// TwinCAT 3 PLC project PackML_Base
// ProgramVersion: 3.1.4023.0
// libraries:
//   PackML State Machine, * (ChrisK)
//   State Pattern PackML, * (ChrisK)
//   Tc2_Standard, * (Beckhoff Automation GmbH)
//   Tc2_System, * (Beckhoff Automation GmbH)
//   Tc3_Module, * (Beckhoff Automation GmbH)
//   Tc3_PackML_V2, * (Beckhoff Automation GmbH)
// project tree:
//   PackML_Method_Sample/ PML_Method_Sample.TcPOU
//   PackML_State_Sample/ Execute_State_Sample.TcPOU, PML_Sample_Class.TcPOU (not stored), Resetting_State_Sample.TcPOU, Starting_State_Sample.TcPOU
//   / PlcTask.TcTTO
//   POUs/ MAIN.TcPOU
// real-time tasks:
//   TASK PlcTask: cycle T#10ms, priority 20, ADS port 350

CONFIGURATION PackML_Base
    RESOURCE PLC ON TwinCAT3
        TASK PlcTask(INTERVAL := T#10ms, PRIORITY := 20);
        PROGRAM MAIN WITH PlcTask : MAIN;
    END_RESOURCE
END_CONFIGURATION

// ---- POUs/MAIN.TcPOU
PROGRAM MAIN
VAR
	pmlbase : PML_StatePattern_Base;
	controlPML : PMLStateMachine;
	subPML1 : PMLStateMachine;
	subPML2 : PMLStateMachine;
	controlpmlmethod : PML_Method_Sample := (PackMLStateMachine := controlPML);
	subpmlmethod1 : PML_Method_Sample := (PackMLStateMachine := subPML1);
	subpmlmethod2 : PML_Method_Sample := (PackMLStateMachine := subPML2);
	binit: BOOL;
	xTest: BOOL;
END_VAR

IF NOT binit THEN
	controlPML.RegisterSubUnit(SubUnit := subPML1);
	controlPML.RegisterSubUnit(SubUnit := subPML2);
	binit := true;
END_IF
controlpmlmethod.Cycle();
subpmlmethod1.Cycle();
subpmlmethod2.Cycle();
controlPML();
subPML1();
subPML2();

IF xTest THEN
	subPML1.PmlModeCommand(Mode := Tc3_PackML_V2.E_PMLProtectedUnitMode.ePMLProtUnitMode_Production);
	subPML2.PmlModeCommand(Mode := Tc3_PackML_V2.E_PMLProtectedUnitMode.ePMLProtUnitMode_Production);
	controlPML.PmlModeCommand(Mode := Tc3_PackML_V2.E_PMLProtectedUnitMode.ePMLProtUnitMode_Production);
	xTest := FALSE;
END_IF

END_PROGRAM

// ---- PackML_Method_Sample/PML_Method_Sample.TcPOU
FUNCTION_BLOCK PML_Method_Sample EXTENDS PML_Method_Base
VAR_INPUT
END_VAR
VAR_OUTPUT
END_VAR
VAR
	ResetMachine : BOOL;
	StartMachine : BOOL;
END_VAR

SUPER^();

METHOD PROTECTED Idle : BOOL
VAR_INPUT
END_VAR
IF StartMachine THEN
	ipackml.PmlStateCommand(Command := E_PMLCommand.ePMLCommand_Start);
END_IF
END_METHOD

METHOD PROTECTED Stopped : BOOL
VAR_INPUT
END_VAR
IF ResetMachine THEN
	ipackml.PmlStateCommand(Command := E_PMLCommand.ePMLCommand_Reset);
END_IF
END_METHOD

END_FUNCTION_BLOCK

// ---- PackML_State_Sample/Execute_State_Sample.TcPOU
FUNCTION_BLOCK Execute_State_Sample  IMPLEMENTS ITF_State
VAR_INPUT
END_VAR
VAR_OUTPUT
END_VAR
VAR
	pPML_Base : POINTER TO PML_StatePattern_Base;
	_stateMachine : IPmlStateMachine;
	bShutdown : BOOL;	
END_VAR

METHOD Cycle : BOOL
VAR_INPUT
END_VAR
IF bShutdown THEN
	pPML_Base^.SetState(pPML_Base^.aborting);
	_stateMachine.PmlStateCommand(Command := E_PMLCommand.ePMLCommand_Abort);
END_IF
END_METHOD

METHOD FB_init : BOOL
VAR_INPUT
	bInitRetains : BOOL; // if TRUE, the retain variables are initialized (warm start / cold start)
	bInCopyCode : BOOL;  // if TRUE, the instance afterwards gets moved into the copy code (online change)
	pPML_Base : POINTER TO PML_StatePattern_Base;
	statemachine : IPmlStateMachine;
END_VAR
_stateMachine := statemachine;
THIS^.pPML_Base := pPML_Base;
END_METHOD

END_FUNCTION_BLOCK

// ---- PackML_State_Sample/Resetting_State_Sample.TcPOU
FUNCTION_BLOCK Resetting_State_Sample  IMPLEMENTS ITF_State
VAR_INPUT
END_VAR
VAR_OUTPUT
END_VAR
VAR
	pPML_Base : POINTER TO PML_StatePattern_Base;
	_stateMachine : IPmlStateMachine;
	bResetComplete : BOOL;
END_VAR

METHOD Cycle : BOOL
VAR_INPUT
END_VAR
IF bResetComplete THEN
	_stateMachine.SetStateComplete();
	pPML_Base^.SetState(pPML_Base^.idle);
END_IF
END_METHOD

METHOD FB_init : BOOL
VAR_INPUT
	bInitRetains : BOOL; // if TRUE, the retain variables are initialized (warm start / cold start)
	bInCopyCode : BOOL;  // if TRUE, the instance afterwards gets moved into the copy code (online change)
	pPML_Base : POINTER TO PML_StatePattern_Base;
	statemachine : IPmlStateMachine;
END_VAR
_stateMachine := statemachine;
THIS^.pPML_Base := pPML_Base;
END_METHOD

END_FUNCTION_BLOCK

// ---- PackML_State_Sample/Starting_State_Sample.TcPOU
FUNCTION_BLOCK Starting_State_Sample  IMPLEMENTS ITF_State
VAR_INPUT
END_VAR
VAR_OUTPUT
END_VAR
VAR
	pPML_Base : POINTER TO PML_StatePattern_Base;
	_stateMachine : IPmlStateMachine;
	bRun: BOOL;
END_VAR

METHOD Cycle : BOOL
VAR_INPUT
END_VAR
IF bRun THEN
	_stateMachine.SetStateComplete();
	pPML_Base^.SetState(pPML_Base^.execute);
END_IF
END_METHOD

METHOD FB_init : BOOL
VAR_INPUT
	bInitRetains : BOOL; // if TRUE, the retain variables are initialized (warm start / cold start)
	bInCopyCode : BOOL;  // if TRUE, the instance afterwards gets moved into the copy code (online change)
	pPML_Base : POINTER TO PML_StatePattern_Base;
	statemachine : IPmlStateMachine;
END_VAR
_stateMachine := statemachine;
THIS^.pPML_Base := pPML_Base;
END_METHOD

END_FUNCTION_BLOCK
